(* Logix 5000 project; controller Thurs_Lab2 vendor 1 type 14 code 156 rev 30.11; software revision 30.00; part 5 of 5 *)
(* tags used below, declared in another part *)
   AUTO : BOOL;
   CYL1_EXT_4_TEST : BOOL;
   CYL1_EXT_PX : BOOL;
   CYL1_RET_4_TEST : BOOL;
   CYL1_RET_PX : BOOL;
   EXTEND : TIMER;
   GOOD_PART : BOOL;
   HOLE_DEPTH_MAX : DINT;
   HOLE_DEPTH_MIN : DINT;
   HOLE_SHALLOW_MAX : DINT;
   HOLE_SHALLOW_MIN : DINT;
   OP5_STATIC_GOOD : BOOL;
   OP5_STATIC_OVER : BOOL;
   OP5_STATIC_REJECT : BOOL;
   OP5_STATIC_UNDER : BOOL;
   OP5_STOP : BOOL;
   OPERATION_5_OVER : BOOL;
   OPERATION_5_REJECT : BOOL;
   OPERATION_5_UNDER : BOOL;
   OPERATION_DONE : DINT;
   OPERATION_OFF : DINT;
   PB3 : BOOL;
   PREVENT_FAULT_5 : DINT;
   PV_HOLE_TOO_DEEP : DINT;
   PV_HOLE_TOO_SHALLOW : DINT;
   RESET : BOOL;
   RESET_OVER_5 : BOOL;
   RESET_REJECT_5 : BOOL;
   RESET_UNDER_5 : BOOL;
   SEQ_EN : BOOL;
   SETTLE5 : TIMER;
   START_SIGNAL : BOOL;
   STEP : DINT;
   Timer : TIMER;
(* MainProgram, continued *)

ROUTINE TEST   (* ladder *)
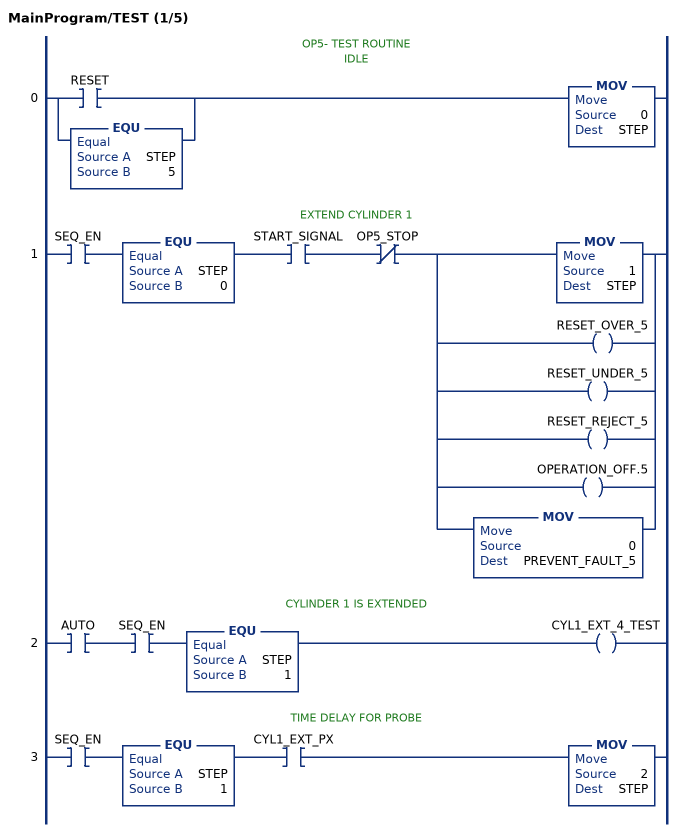
   // OP5- TEST ROUTINE
   // IDLE
   0: [XIC(RESET) ,EQU(STEP,5) ]MOV(0,STEP);
   // EXTEND CYLINDER 1
   1: XIC(SEQ_EN)EQU(STEP,0)XIC(START_SIGNAL)XIO(OP5_STOP)[MOV(1,STEP) ,OTE(RESET_OVER_5) ,OTE(RESET_UNDER_5) ,OTE(RESET_REJECT_5) ,OTE(OPERATION_OFF.5) ,MOV(0,PREVENT_FAULT_5) ];
   // CYLINDER 1 IS EXTENDED
   2: XIC(AUTO)XIC(SEQ_EN)EQU(STEP,1)OTE(CYL1_EXT_4_TEST);
   // TIME DELAY FOR PROBE
   3: XIC(SEQ_EN)EQU(STEP,1)XIC(CYL1_EXT_PX)MOV(2,STEP);
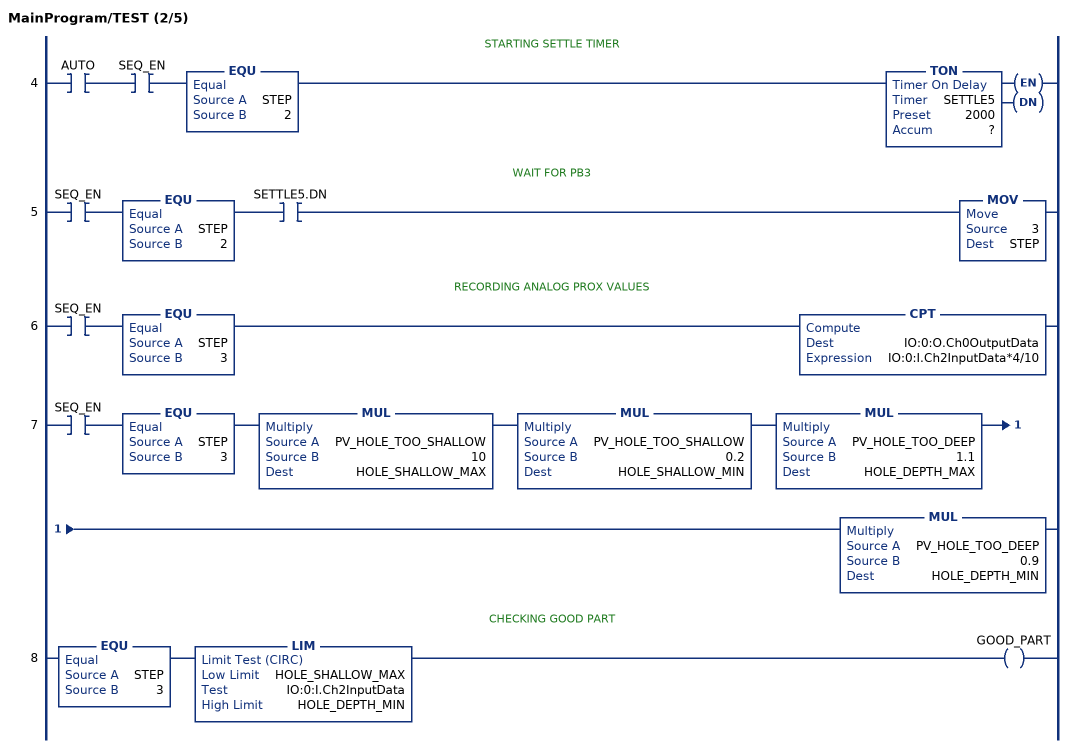
   // STARTING SETTLE TIMER
   4: XIC(AUTO)XIC(SEQ_EN)EQU(STEP,2)TON(SETTLE5,?,?);
   // WAIT FOR PB3
   5: XIC(SEQ_EN)EQU(STEP,2)XIC(SETTLE5.DN)MOV(3,STEP);
   // RECORDING ANALOG PROX VALUES
   6: XIC(SEQ_EN)EQU(STEP,3)CPT(IO:0:O.Ch0OutputData,IO:0:I.Ch2InputData*4/10);
   7: XIC(SEQ_EN)EQU(STEP,3)MUL(PV_HOLE_TOO_SHALLOW,10,HOLE_SHALLOW_MAX)MUL(PV_HOLE_TOO_SHALLOW,0.2,HOLE_SHALLOW_MIN)MUL(PV_HOLE_TOO_DEEP,1.1,HOLE_DEPTH_MAX)MUL(PV_HOLE_TOO_DEEP,0.9,HOLE_DEPTH_MIN);
   // CHECKING GOOD PART
   8: EQU(STEP,3)LIM(HOLE_SHALLOW_MAX,IO:0:I.Ch2InputData,HOLE_DEPTH_MIN)OTE(GOOD_PART);
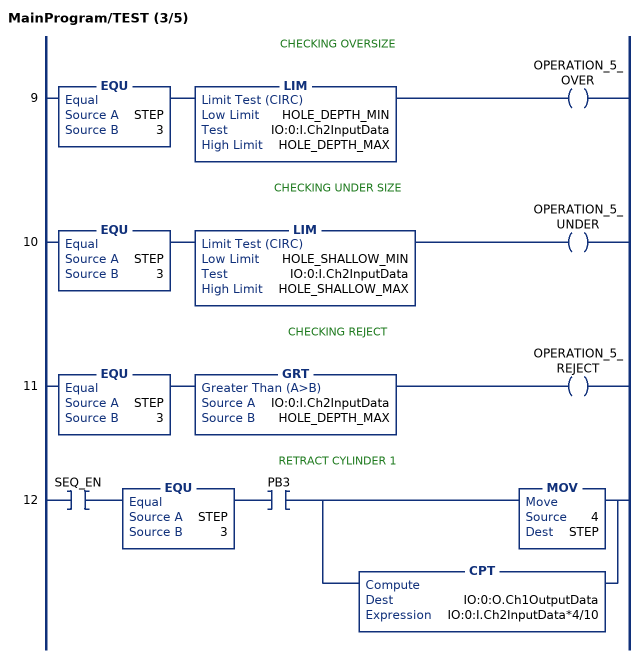
   // CHECKING OVERSIZE
   9: EQU(STEP,3)LIM(HOLE_DEPTH_MIN,IO:0:I.Ch2InputData,HOLE_DEPTH_MAX)OTE(OPERATION_5_OVER);
   // CHECKING UNDER SIZE
   10: EQU(STEP,3)LIM(HOLE_SHALLOW_MIN,IO:0:I.Ch2InputData,HOLE_SHALLOW_MAX)OTE(OPERATION_5_UNDER);
   // CHECKING REJECT
   11: EQU(STEP,3)GRT(IO:0:I.Ch2InputData,HOLE_DEPTH_MAX)OTE(OPERATION_5_REJECT);
   // RETRACT CYLINDER 1
   12: XIC(SEQ_EN)EQU(STEP,3)XIC(PB3)[MOV(4,STEP) ,CPT(IO:0:O.Ch1OutputData,IO:0:I.Ch2InputData*4/10) ];
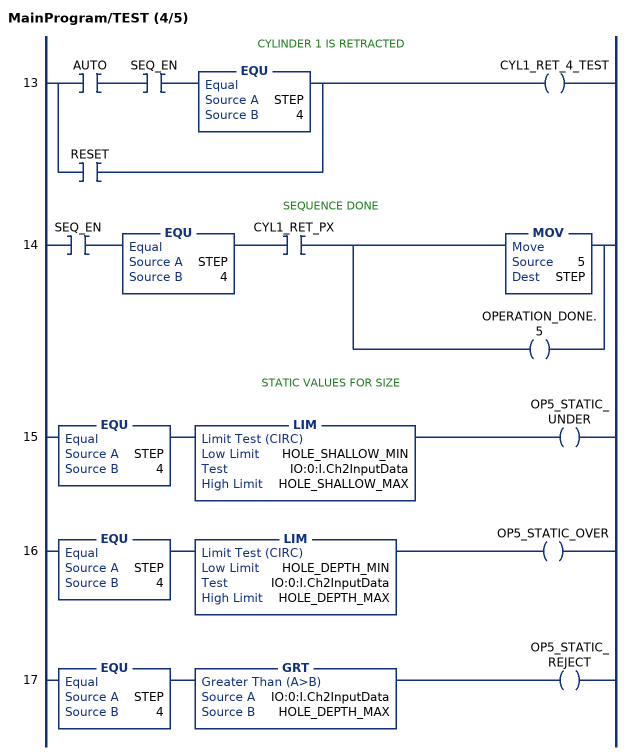
   // CYLINDER 1 IS RETRACTED
   13: [XIC(AUTO) XIC(SEQ_EN) EQU(STEP,4) ,XIC(RESET) ]OTE(CYL1_RET_4_TEST);
   // SEQUENCE DONE
   14: XIC(SEQ_EN)EQU(STEP,4)XIC(CYL1_RET_PX)[MOV(5,STEP) ,OTE(OPERATION_DONE.5) ];
   // STATIC VALUES FOR SIZE
   15: EQU(STEP,4)LIM(HOLE_SHALLOW_MIN,IO:0:I.Ch2InputData,HOLE_SHALLOW_MAX)OTE(OP5_STATIC_UNDER);
   16: EQU(STEP,4)LIM(HOLE_DEPTH_MIN,IO:0:I.Ch2InputData,HOLE_DEPTH_MAX)OTE(OP5_STATIC_OVER);
   17: EQU(STEP,4)GRT(IO:0:I.Ch2InputData,HOLE_DEPTH_MAX)OTE(OP5_STATIC_REJECT);
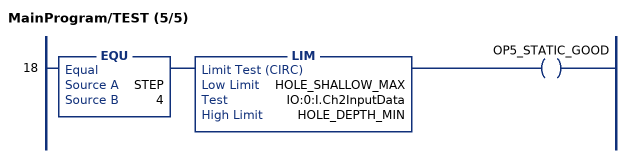
   18: EQU(STEP,4)LIM(HOLE_SHALLOW_MAX,IO:0:I.Ch2InputData,HOLE_DEPTH_MIN)OTE(OP5_STATIC_GOOD);
END_ROUTINE
END_PROGRAM
